TYPE "UDT_SUCDataAssembly"
VERSION : 0.1
   STRUCT
      tag_name : String;
      tag_description : String;
   END_STRUCT;

END_TYPE

